(* CoDeSys 2.3 export: STEAMVALVE_KD2.EXP *)

(* POU PRG/SteamValve_KD2, ST *)
PROGRAM SteamValve_KD2
VAR
END_VAR
	IF NOT KD2.SteamValve.xMode_AUTO THEN
		;
	END_IF;
END_PROGRAM
